(* PLC project Unnamed, Unknown Unnamed 1 *)
(* stored: creationDateTime 2026-05-27T00:32:00, modificationDateTime 2026-05-27T00:32:00 *)

PROGRAM main
  VAR
    bt_start_t1 AT %IX0.0 : BOOL;
    bt_stop_t1 AT %IX0.1 : BOOL;
    led_start_t1 AT %QX0.0 : BOOL;
  END_VAR

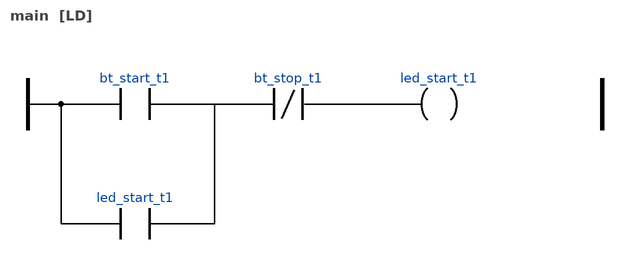
(* LD diagram, written out as Structured Text *)
led_start_t1 := (bt_start_t1 OR led_start_t1) AND NOT bt_stop_t1;
END_PROGRAM

CONFIGURATION Config0
  RESOURCE Res0 ON PLC
    TASK task0(INTERVAL := T#20ms, PRIORITY := 1);
    PROGRAM instance0 WITH task0 : main;
  END_RESOURCE
END_CONFIGURATION
